// TIA Portal project "Separating_Station" (V15.1)

(* hardware
DEVICE "S7-1200 station_1"  S7-1200 Station
   slot 0: "Rack_0"  S7-1200 Rack  Rack  V1.0
   slot 1: "PLC_1"  CPU 1212C AC/DC/Rly  6ES7 212-1BE40-0XB0  V4.3
*)

// ===== PLC "PLC_1"  CPU 1212C AC/DC/Rly =====

VAR_GLOBAL   // PLC tag table "Default tag table"
   "System_Byte" AT %MB1 : Byte;
   "FirstScan" AT %M1.0 : Bool;
   "DiagStatusUpdate" AT %M1.1 : Bool;
   "AlwaysTRUE" AT %M1.2 : Bool;
   "AlwaysFALSE" AT %M1.3 : Bool;
   "Clock_Byte" AT %MB0 : Byte;
   "Clock_10Hz" AT %M0.0 : Bool;
   "Clock_5Hz" AT %M0.1 : Bool;
   "Clock_2.5Hz" AT %M0.2 : Bool;
   "Clock_2Hz" AT %M0.3 : Bool;
   "Clock_1.25Hz" AT %M0.4 : Bool;
   "Clock_1Hz" AT %M0.5 : Bool;
   "Clock_0.625Hz" AT %M0.6 : Bool;
   "Clock_0.5Hz" AT %M0.7 : Bool;
   "Start" AT %I21.0 : Bool;
   "Stop" AT %I21.1 : Bool;
   "Entry_Conveyor_1" AT %Q20.0 : Bool;
   "SQ_Pusher_1_Front" AT %I20.2 : Bool;
   "SQ_Pusher_1_Back" AT %I20.3 : Bool;
   "Vision_Sensor_1" AT %IW100 : Int;
   "Vision_Sensor_2" AT %IW102 : Int;
   "Entry_Conveyor_2" AT %Q20.1 : Bool;
   "SQ_Pusher_2_Back" AT %I20.6 : Bool;
   "SQ_1" AT %I20.0 : Bool;
   "SQ_2" AT %I20.1 : Bool;
   "Conveyor_1" AT %Q20.2 : Bool;
   "Conveyor_2" AT %Q20.3 : Bool;
   "At_Pusher_1_Exit" AT %I20.4 : Bool;
   "At_Pusher_2_Exit" AT %I20.7 : Bool;
   "Pusher_1" AT %Q20.4 : Bool;
   "Pusher_2" AT %Q20.5 : Bool;
   "SQ_Pusher_2_Front" AT %I20.5 : Bool;
   "Tag_2" AT %I21.2 : Bool;
END_VAR

DATA_BLOCK "Ist_Separating_Station"   // DB1
{ S7_Optimized_Access := 'TRUE' }
AUTHOR : Rackso
VERSION : 0.1
// stored: InstanceOfName Separating_Station
"Separating_Station"
BEGIN
END_DATA_BLOCK

DATA_BLOCK "Edge"   // DB3
{ S7_Optimized_Access := 'TRUE' }
AUTHOR : Rackso
VERSION : 0.1
   VAR
      Negative_Edge : Array[0..15] of Bool;
      Positve_Edge : Array[0..15] of Bool;
   END_VAR
BEGIN
END_DATA_BLOCK

FUNCTION_BLOCK "Separating_Station"   // FB2, LAD
{ S7_Optimized_Access := 'TRUE' }
AUTHOR : Rackso
VERSION : 0.1
   VAR_INPUT
      Sensor_1 : Bool;   // At "Entry conveyor_1" exit
      Sensor_2 : Bool;   // At "Entry conveyor_2" exit
      Pusher_1_front : Bool;   // Extended pusher_1
      Pusher_1_back : Bool;   // Retracted pusher_1
      At_pusher_1_exit : Bool;   // Counter_1
      Pusher_2_front : Bool;   // Extended pusher_2
      Pusher_2_back : Bool;   // Retracted pusher_2
      At_pusher_2_exit : Bool;   // Counter_2
      Start : Bool;
      Stop : Bool;
      FactoryIO_Running : Bool;
      EM_Stop : Bool;
      PEW_Vision_sensor_1 : Int;   // Recognizes raw material "colors" 1=blue, 4=green
      PEW_Vision_sensor_2 : Int;   // Recognizes raw material "colors" 1=blue, 4=green
   END_VAR
   VAR_OUTPUT
      Entry_conveyor_1 : Bool;
      Entry_conveyor_2 : Bool;
      Conveyor_1 : Bool;
      Conveyor_2 : Bool;
      Pusher_1 : Bool;
      Pusher_2 : Bool;
      Emiter_1 : Bool;
      Emiter_2 : Bool;
      Start_light : Bool;
      Stop_light : Bool;
      Reset_light : Bool;
      Counter_1 : Bool;
      Counter_2 : Bool;
   END_VAR
   VAR
      Run_Process : Bool;
      X_Sensor_1 : Bool;
      X_Sensor_2 : Bool;
      Event_1 : Bool;
      X_At_Pusher_1_Exit : Bool;
      Aux_1 : Bool;
      Aux_2 : Bool;
      Event_2 : Bool;
      Event_3 : Bool;
      Event_4 : Bool;
      X_Pusher_1_Back : Bool;
      X_Pusher_2_Back : Bool;
      Event_5 : Bool;
      Event_6 : Bool;
      Event_7 : Bool;
      X_At_Pusher_2_Exit : Bool;
      Aux_Retract_1 : Bool;
      Y1 : Bool;
      Y2 : Bool;
      Aux_Retract_2 : Bool;
      Y3 : Bool;
      Aux_Retract_3 : Bool;
      Aux_1_Conveyor : Bool;
      EN_1_Conveyor_1 : Bool;
      CZ1 : Bool;
      EN_1_Conveyor_2 : Bool;
      Aux_2_Conveyor : Bool;
      EN_2_Conveyor_1 : Bool;
      CZ2 : Bool;
      EN_2_Conveyor_2 : Bool;
      Aux_3_Conveyor : Bool;
      CZ3 : Bool;
      EN_3_Conveyor_1 : Bool;
      EN_3_Conveyor_2 : Bool;
      CZ4 : Bool;
      EN_4_Conveyor_1 : Bool;
      EN_4_Conveyor_2 : Bool;
      Event_8 : Bool;
      Aux_Pusher_1 : Bool;
      Aux_Pusher_2 : Bool;
   END_VAR
   VAR_TEMP   // added for the SCL form of the ladder/FBD networks
      _w1 : Bool;
      _w2 : Bool;
      _w3 : Bool;
      _w4 : Bool;
      _w5 : Bool;
      _w6 : Bool;
      _w7 : Bool;
      _w8 : Bool;
      _w9 : Bool;
      _w10 : Bool;
      _w11 : Bool;
      _w12 : Bool;
      _w13 : Bool;
   END_VAR
BEGIN

REGION Network 1: Start Process
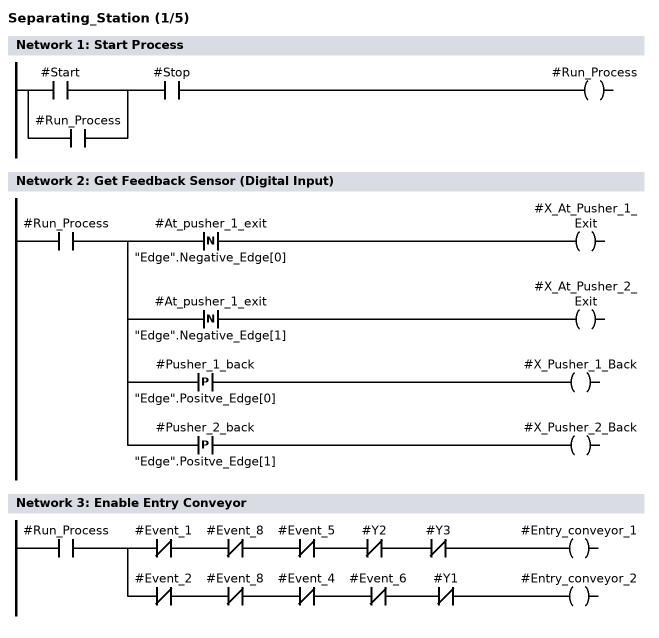
   RUNG wire#powerrail
      Contact( #Start )
      wire#w1
      Contact( #Stop )
      Coil( #Run_Process )
   END_RUNG
   RUNG wire#powerrail
      Contact( #Run_Process )
   END_RUNG wire#w1
   // the same network as SCL:
   #Run_Process := (#Start OR #Run_Process) AND #Stop;
END_REGION

REGION Network 2: Get Feedback Sensor (Digital Input)
   RUNG wire#powerrail
      Contact( #Run_Process )
      wire#w1
      N_Contact(operand := #At_pusher_1_exit, bit := "Edge".Negative_Edge[0])
      Coil( #X_At_Pusher_1_Exit )
   END_RUNG
   RUNG wire#w1
      N_Contact(operand := #At_pusher_1_exit, bit := "Edge".Negative_Edge[1])
      Coil( #X_At_Pusher_2_Exit )
   END_RUNG
   RUNG wire#w1
      P_Contact(operand := #Pusher_1_back, bit := "Edge".Positve_Edge[0])
      Coil( #X_Pusher_1_Back )
   END_RUNG
   RUNG wire#w1
      P_Contact(operand := #Pusher_2_back, bit := "Edge".Positve_Edge[1])
      Coil( #X_Pusher_2_Back )
   END_RUNG
   // the same network as SCL:
   #_w1 := #Run_Process AND NOT #At_pusher_1_exit AND "Edge".Negative_Edge[0];   // falling edge of #At_pusher_1_exit
   "Edge".Negative_Edge[0] := #At_pusher_1_exit;
   #X_At_Pusher_1_Exit := #_w1;
   #_w2 := #Run_Process AND NOT #At_pusher_1_exit AND "Edge".Negative_Edge[1];   // falling edge of #At_pusher_1_exit
   "Edge".Negative_Edge[1] := #At_pusher_1_exit;
   #X_At_Pusher_2_Exit := #_w2;
   #_w3 := #Run_Process AND #Pusher_1_back AND NOT "Edge".Positve_Edge[0];   // rising edge of #Pusher_1_back
   "Edge".Positve_Edge[0] := #Pusher_1_back;
   #X_Pusher_1_Back := #_w3;
   #_w4 := #Run_Process AND #Pusher_2_back AND NOT "Edge".Positve_Edge[1];   // rising edge of #Pusher_2_back
   "Edge".Positve_Edge[1] := #Pusher_2_back;
   #X_Pusher_2_Back := #_w4;
END_REGION

REGION Network 3: Enable Entry Conveyor
   RUNG wire#powerrail
      Contact( #Run_Process )
      wire#w1
      I_Contact( #Event_1 )
      I_Contact( #Event_8 )
      I_Contact( #Event_5 )
      I_Contact( #Y2 )
      I_Contact( #Y3 )
      Coil( #Entry_conveyor_1 )
   END_RUNG
   RUNG wire#w1
      I_Contact( #Event_2 )
      I_Contact( #Event_8 )
      I_Contact( #Event_4 )
      I_Contact( #Event_6 )
      I_Contact( #Y1 )
      Coil( #Entry_conveyor_2 )
   END_RUNG
   // the same network as SCL:
   #Entry_conveyor_1 := #Run_Process AND NOT #Event_1 AND NOT #Event_8 AND NOT #Event_5 AND NOT #Y2 AND NOT #Y3;
   #Entry_conveyor_2 := #Run_Process AND NOT #Event_2 AND NOT #Event_8 AND NOT #Event_4 AND NOT #Event_6 AND NOT #Y1;
END_REGION

REGION Network 4: Get Feedback Sensor Analog Input)
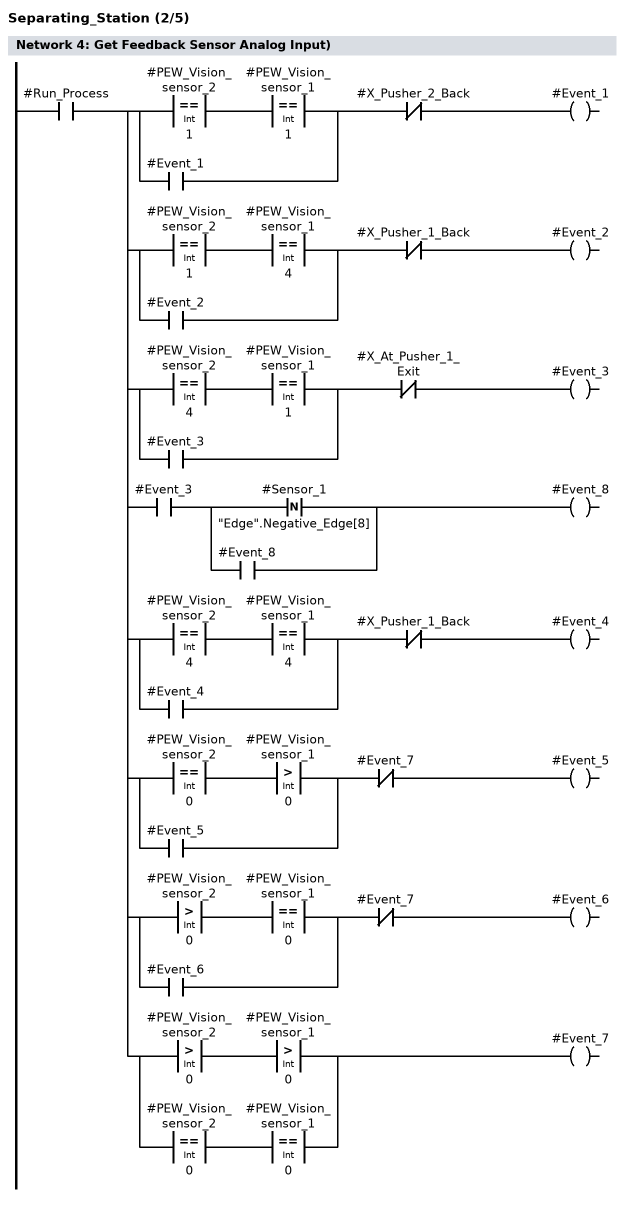
   RUNG wire#powerrail
      Contact( #Run_Process )
      wire#w1
      { S7_Templates := "SrcType := Int" } EQ_Contact(in1 := #PEW_Vision_sensor_2, in2 := 1)
      { S7_Templates := "SrcType := Int" } EQ_Contact(in1 := #PEW_Vision_sensor_1, in2 := 1)
      wire#w2
      I_Contact( #X_Pusher_2_Back )
      Coil( #Event_1 )
   END_RUNG
   RUNG wire#w1
      Contact( #Event_1 )
   END_RUNG wire#w2
   RUNG wire#w1
      { S7_Templates := "SrcType := Int" } EQ_Contact(in1 := #PEW_Vision_sensor_2, in2 := 1)
      { S7_Templates := "SrcType := Int" } EQ_Contact(in1 := #PEW_Vision_sensor_1, in2 := 4)
      wire#w3
      I_Contact( #X_Pusher_1_Back )
      Coil( #Event_2 )
   END_RUNG
   RUNG wire#w1
      Contact( #Event_2 )
   END_RUNG wire#w3
   RUNG wire#w1
      { S7_Templates := "SrcType := Int" } EQ_Contact(in1 := #PEW_Vision_sensor_2, in2 := 4)
      { S7_Templates := "SrcType := Int" } EQ_Contact(in1 := #PEW_Vision_sensor_1, in2 := 1)
      wire#w4
      I_Contact( #X_At_Pusher_1_Exit )
      Coil( #Event_3 )
   END_RUNG
   RUNG wire#w1
      Contact( #Event_3 )
   END_RUNG wire#w4
   RUNG wire#w1
      Contact( #Event_3 )
      wire#w5
      N_Contact(operand := #Sensor_1, bit := "Edge".Negative_Edge[8])
      wire#w6
      Coil( #Event_8 )
   END_RUNG
   RUNG wire#w5
      Contact( #Event_8 )
   END_RUNG wire#w6
   RUNG wire#w1
      { S7_Templates := "SrcType := Int" } EQ_Contact(in1 := #PEW_Vision_sensor_2, in2 := 4)
      { S7_Templates := "SrcType := Int" } EQ_Contact(in1 := #PEW_Vision_sensor_1, in2 := 4)
      wire#w7
      I_Contact( #X_Pusher_1_Back )
      Coil( #Event_4 )
   END_RUNG
   RUNG wire#w1
      Contact( #Event_4 )
   END_RUNG wire#w7
   RUNG wire#w1
      { S7_Templates := "SrcType := Int" } EQ_Contact(in1 := #PEW_Vision_sensor_2, in2 := 0)
      { S7_Templates := "SrcType := Int" } GT_Contact(in1 := #PEW_Vision_sensor_1, in2 := 0)
      wire#w8
      I_Contact( #Event_7 )
      Coil( #Event_5 )
   END_RUNG
   RUNG wire#w1
      Contact( #Event_5 )
   END_RUNG wire#w8
   RUNG wire#w1
      { S7_Templates := "SrcType := Int" } GT_Contact(in1 := #PEW_Vision_sensor_2, in2 := 0)
      { S7_Templates := "SrcType := Int" } EQ_Contact(in1 := #PEW_Vision_sensor_1, in2 := 0)
      wire#w9
      I_Contact( #Event_7 )
      Coil( #Event_6 )
   END_RUNG
   RUNG wire#w1
      Contact( #Event_6 )
   END_RUNG wire#w9
   RUNG wire#w1
      { S7_Templates := "SrcType := Int" } GT_Contact(in1 := #PEW_Vision_sensor_2, in2 := 0)
      { S7_Templates := "SrcType := Int" } GT_Contact(in1 := #PEW_Vision_sensor_1, in2 := 0)
      wire#w10
      Coil( #Event_7 )
   END_RUNG
   RUNG wire#w1
      { S7_Templates := "SrcType := Int" } EQ_Contact(in1 := #PEW_Vision_sensor_2, in2 := 0)
      { S7_Templates := "SrcType := Int" } EQ_Contact(in1 := #PEW_Vision_sensor_1, in2 := 0)
   END_RUNG wire#w10
   // the same network as SCL:
   #Event_1 := #Run_Process AND (((#PEW_Vision_sensor_2 = 1) AND (#PEW_Vision_sensor_1 = 1)) OR #Event_1) AND NOT #X_Pusher_2_Back;
   #Event_2 := #Run_Process AND (((#PEW_Vision_sensor_2 = 1) AND (#PEW_Vision_sensor_1 = 4)) OR #Event_2) AND NOT #X_Pusher_1_Back;
   #Event_3 := #Run_Process AND (((#PEW_Vision_sensor_2 = 4) AND (#PEW_Vision_sensor_1 = 1)) OR #Event_3) AND NOT #X_At_Pusher_1_Exit;
   #_w1 := #Run_Process AND #Event_3 AND NOT #Sensor_1 AND "Edge".Negative_Edge[8];   // falling edge of #Sensor_1
   "Edge".Negative_Edge[8] := #Sensor_1;
   #Event_8 := #_w1 OR (#Run_Process AND #Event_3 AND #Event_8);
   #Event_4 := #Run_Process AND (((#PEW_Vision_sensor_2 = 4) AND (#PEW_Vision_sensor_1 = 4)) OR #Event_4) AND NOT #X_Pusher_1_Back;
   #Event_5 := #Run_Process AND (((#PEW_Vision_sensor_2 = 0) AND (#PEW_Vision_sensor_1 > 0)) OR #Event_5) AND NOT #Event_7;
   #Event_6 := #Run_Process AND (((#PEW_Vision_sensor_2 > 0) AND (#PEW_Vision_sensor_1 = 0)) OR #Event_6) AND NOT #Event_7;
   #Event_7 := #Run_Process AND (((#PEW_Vision_sensor_2 > 0) AND (#PEW_Vision_sensor_1 > 0)) OR ((#PEW_Vision_sensor_2 = 0) AND (#PEW_Vision_sensor_1 = 0)));
END_REGION

REGION Network 5: Aux Enable Pusher
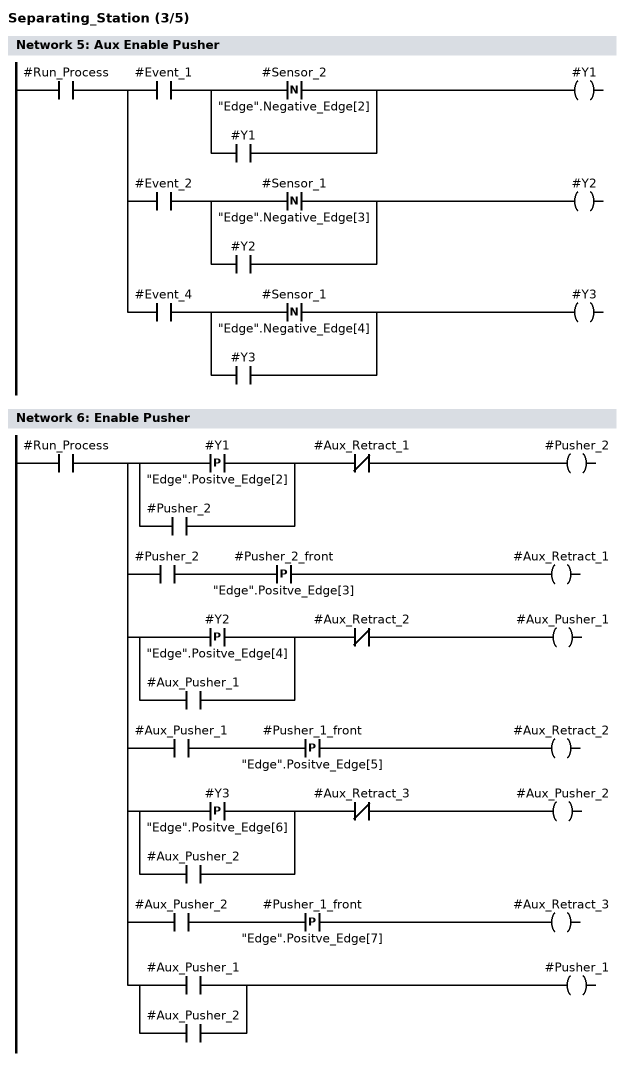
   RUNG wire#powerrail
      Contact( #Run_Process )
      wire#w1
      Contact( #Event_1 )
      wire#w2
      N_Contact(operand := #Sensor_2, bit := "Edge".Negative_Edge[2])
      wire#w3
      Coil( #Y1 )
   END_RUNG
   RUNG wire#w2
      Contact( #Y1 )
   END_RUNG wire#w3
   RUNG wire#w1
      Contact( #Event_2 )
      wire#w4
      N_Contact(operand := #Sensor_1, bit := "Edge".Negative_Edge[3])
      wire#w5
      Coil( #Y2 )
   END_RUNG
   RUNG wire#w4
      Contact( #Y2 )
   END_RUNG wire#w5
   RUNG wire#w1
      Contact( #Event_4 )
      wire#w6
      N_Contact(operand := #Sensor_1, bit := "Edge".Negative_Edge[4])
      wire#w7
      Coil( #Y3 )
   END_RUNG
   RUNG wire#w6
      Contact( #Y3 )
   END_RUNG wire#w7
   // the same network as SCL:
   #_w1 := #Run_Process AND #Event_1 AND NOT #Sensor_2 AND "Edge".Negative_Edge[2];   // falling edge of #Sensor_2
   "Edge".Negative_Edge[2] := #Sensor_2;
   #Y1 := #_w1 OR (#Run_Process AND #Event_1 AND #Y1);
   #_w2 := #Run_Process AND #Event_2 AND NOT #Sensor_1 AND "Edge".Negative_Edge[3];   // falling edge of #Sensor_1
   "Edge".Negative_Edge[3] := #Sensor_1;
   #Y2 := #_w2 OR (#Run_Process AND #Event_2 AND #Y2);
   #_w3 := #Run_Process AND #Event_4 AND NOT #Sensor_1 AND "Edge".Negative_Edge[4];   // falling edge of #Sensor_1
   "Edge".Negative_Edge[4] := #Sensor_1;
   #Y3 := #_w3 OR (#Run_Process AND #Event_4 AND #Y3);
END_REGION

REGION Network 6: Enable Pusher
   RUNG wire#powerrail
      Contact( #Run_Process )
      wire#w1
      P_Contact(operand := #Y1, bit := "Edge".Positve_Edge[2])
      wire#w2
      I_Contact( #Aux_Retract_1 )
      Coil( #Pusher_2 )
   END_RUNG
   RUNG wire#w1
      Contact( #Pusher_2 )
   END_RUNG wire#w2
   RUNG wire#w1
      Contact( #Pusher_2 )
      P_Contact(operand := #Pusher_2_front, bit := "Edge".Positve_Edge[3])
      Coil( #Aux_Retract_1 )
   END_RUNG
   RUNG wire#w1
      P_Contact(operand := #Y2, bit := "Edge".Positve_Edge[4])
      wire#w3
      I_Contact( #Aux_Retract_2 )
      Coil( #Aux_Pusher_1 )
   END_RUNG
   RUNG wire#w1
      Contact( #Aux_Pusher_1 )
   END_RUNG wire#w3
   RUNG wire#w1
      Contact( #Aux_Pusher_1 )
      P_Contact(operand := #Pusher_1_front, bit := "Edge".Positve_Edge[5])
      Coil( #Aux_Retract_2 )
   END_RUNG
   RUNG wire#w1
      P_Contact(operand := #Y3, bit := "Edge".Positve_Edge[6])
      wire#w4
      I_Contact( #Aux_Retract_3 )
      Coil( #Aux_Pusher_2 )
   END_RUNG
   RUNG wire#w1
      Contact( #Aux_Pusher_2 )
   END_RUNG wire#w4
   RUNG wire#w1
      Contact( #Aux_Pusher_2 )
      P_Contact(operand := #Pusher_1_front, bit := "Edge".Positve_Edge[7])
      Coil( #Aux_Retract_3 )
   END_RUNG
   RUNG wire#w1
      Contact( #Aux_Pusher_1 )
      wire#w5
      Coil( #Pusher_1 )
   END_RUNG
   RUNG wire#w1
      Contact( #Aux_Pusher_2 )
   END_RUNG wire#w5
   // the same network as SCL:
   #_w1 := #Run_Process AND #Y1 AND NOT "Edge".Positve_Edge[2];   // rising edge of #Y1
   "Edge".Positve_Edge[2] := #Y1;
   #Pusher_2 := (#_w1 OR (#Run_Process AND #Pusher_2)) AND NOT #Aux_Retract_1;
   #_w2 := #Run_Process AND #Pusher_2 AND #Pusher_2_front AND NOT "Edge".Positve_Edge[3];   // rising edge of #Pusher_2_front
   "Edge".Positve_Edge[3] := #Pusher_2_front;
   #Aux_Retract_1 := #_w2;
   #_w3 := #Run_Process AND #Y2 AND NOT "Edge".Positve_Edge[4];   // rising edge of #Y2
   "Edge".Positve_Edge[4] := #Y2;
   #Aux_Pusher_1 := (#_w3 OR (#Run_Process AND #Aux_Pusher_1)) AND NOT #Aux_Retract_2;
   #_w4 := #Run_Process AND #Aux_Pusher_1 AND #Pusher_1_front AND NOT "Edge".Positve_Edge[5];   // rising edge of #Pusher_1_front
   "Edge".Positve_Edge[5] := #Pusher_1_front;
   #Aux_Retract_2 := #_w4;
   #_w5 := #Run_Process AND #Y3 AND NOT "Edge".Positve_Edge[6];   // rising edge of #Y3
   "Edge".Positve_Edge[6] := #Y3;
   #Aux_Pusher_2 := (#_w5 OR (#Run_Process AND #Aux_Pusher_2)) AND NOT #Aux_Retract_3;
   #_w6 := #Run_Process AND #Aux_Pusher_2 AND #Pusher_1_front AND NOT "Edge".Positve_Edge[7];   // rising edge of #Pusher_1_front
   "Edge".Positve_Edge[7] := #Pusher_1_front;
   #Aux_Retract_3 := #_w6;
   #Pusher_1 := #Run_Process AND (#Aux_Pusher_1 OR #Aux_Pusher_2);
END_REGION

REGION Network 7: Aux Enbale Conveyor
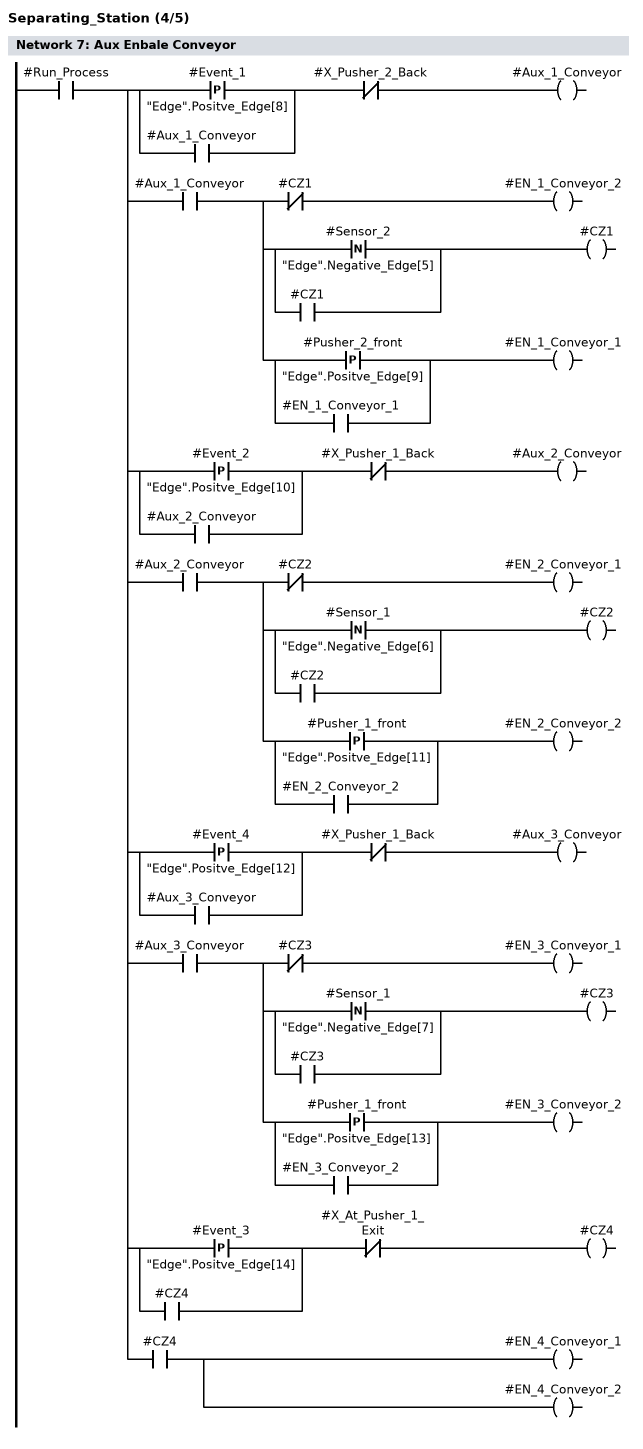
   RUNG wire#powerrail
      Contact( #Run_Process )
      wire#w1
      P_Contact(operand := #Event_1, bit := "Edge".Positve_Edge[8])
      wire#w2
      I_Contact( #X_Pusher_2_Back )
      Coil( #Aux_1_Conveyor )
   END_RUNG
   RUNG wire#w1
      Contact( #Aux_1_Conveyor )
   END_RUNG wire#w2
   RUNG wire#w1
      Contact( #Aux_1_Conveyor )
      wire#w3
      I_Contact( #CZ1 )
      Coil( #EN_1_Conveyor_2 )
   END_RUNG
   RUNG wire#w3
      N_Contact(operand := #Sensor_2, bit := "Edge".Negative_Edge[5])
      wire#w4
      Coil( #CZ1 )
   END_RUNG
   RUNG wire#w3
      Contact( #CZ1 )
   END_RUNG wire#w4
   RUNG wire#w3
      P_Contact(operand := #Pusher_2_front, bit := "Edge".Positve_Edge[9])
      wire#w5
      Coil( #EN_1_Conveyor_1 )
   END_RUNG
   RUNG wire#w3
      Contact( #EN_1_Conveyor_1 )
   END_RUNG wire#w5
   RUNG wire#w1
      P_Contact(operand := #Event_2, bit := "Edge".Positve_Edge[10])
      wire#w6
      I_Contact( #X_Pusher_1_Back )
      Coil( #Aux_2_Conveyor )
   END_RUNG
   RUNG wire#w1
      Contact( #Aux_2_Conveyor )
   END_RUNG wire#w6
   RUNG wire#w1
      Contact( #Aux_2_Conveyor )
      wire#w7
      I_Contact( #CZ2 )
      Coil( #EN_2_Conveyor_1 )
   END_RUNG
   RUNG wire#w7
      N_Contact(operand := #Sensor_1, bit := "Edge".Negative_Edge[6])
      wire#w8
      Coil( #CZ2 )
   END_RUNG
   RUNG wire#w7
      Contact( #CZ2 )
   END_RUNG wire#w8
   RUNG wire#w7
      P_Contact(operand := #Pusher_1_front, bit := "Edge".Positve_Edge[11])
      wire#w9
      Coil( #EN_2_Conveyor_2 )
   END_RUNG
   RUNG wire#w7
      Contact( #EN_2_Conveyor_2 )
   END_RUNG wire#w9
   RUNG wire#w1
      P_Contact(operand := #Event_4, bit := "Edge".Positve_Edge[12])
      wire#w10
      I_Contact( #X_Pusher_1_Back )
      Coil( #Aux_3_Conveyor )
   END_RUNG
   RUNG wire#w1
      Contact( #Aux_3_Conveyor )
   END_RUNG wire#w10
   RUNG wire#w1
      Contact( #Aux_3_Conveyor )
      wire#w11
      I_Contact( #CZ3 )
      Coil( #EN_3_Conveyor_1 )
   END_RUNG
   RUNG wire#w11
      N_Contact(operand := #Sensor_1, bit := "Edge".Negative_Edge[7])
      wire#w12
      Coil( #CZ3 )
   END_RUNG
   RUNG wire#w11
      Contact( #CZ3 )
   END_RUNG wire#w12
   RUNG wire#w11
      P_Contact(operand := #Pusher_1_front, bit := "Edge".Positve_Edge[13])
      wire#w13
      Coil( #EN_3_Conveyor_2 )
   END_RUNG
   RUNG wire#w11
      Contact( #EN_3_Conveyor_2 )
   END_RUNG wire#w13
   RUNG wire#w1
      P_Contact(operand := #Event_3, bit := "Edge".Positve_Edge[14])
      wire#w14
      I_Contact( #X_At_Pusher_1_Exit )
      Coil( #CZ4 )
   END_RUNG
   RUNG wire#w1
      Contact( #CZ4 )
   END_RUNG wire#w14
   RUNG wire#w1
      Contact( #CZ4 )
      wire#w15
      Coil( #EN_4_Conveyor_1 )
   END_RUNG
   RUNG wire#w15
      Coil( #EN_4_Conveyor_2 )
   END_RUNG
   // the same network as SCL:
   #_w1 := #Run_Process AND #Event_1 AND NOT "Edge".Positve_Edge[8];   // rising edge of #Event_1
   "Edge".Positve_Edge[8] := #Event_1;
   #Aux_1_Conveyor := (#_w1 OR (#Run_Process AND #Aux_1_Conveyor)) AND NOT #X_Pusher_2_Back;
   #_w2 := #Run_Process AND #Aux_1_Conveyor;
   #EN_1_Conveyor_2 := #_w2 AND NOT #CZ1;
   #_w3 := #_w2 AND NOT #Sensor_2 AND "Edge".Negative_Edge[5];   // falling edge of #Sensor_2
   "Edge".Negative_Edge[5] := #Sensor_2;
   #CZ1 := #_w3 OR (#_w2 AND #CZ1);
   #_w4 := #_w2 AND #Pusher_2_front AND NOT "Edge".Positve_Edge[9];   // rising edge of #Pusher_2_front
   "Edge".Positve_Edge[9] := #Pusher_2_front;
   #EN_1_Conveyor_1 := #_w4 OR (#_w2 AND #EN_1_Conveyor_1);
   #_w5 := #Run_Process AND #Event_2 AND NOT "Edge".Positve_Edge[10];   // rising edge of #Event_2
   "Edge".Positve_Edge[10] := #Event_2;
   #Aux_2_Conveyor := (#_w5 OR (#Run_Process AND #Aux_2_Conveyor)) AND NOT #X_Pusher_1_Back;
   #_w6 := #Run_Process AND #Aux_2_Conveyor;
   #EN_2_Conveyor_1 := #_w6 AND NOT #CZ2;
   #_w7 := #_w6 AND NOT #Sensor_1 AND "Edge".Negative_Edge[6];   // falling edge of #Sensor_1
   "Edge".Negative_Edge[6] := #Sensor_1;
   #CZ2 := #_w7 OR (#_w6 AND #CZ2);
   #_w8 := #_w6 AND #Pusher_1_front AND NOT "Edge".Positve_Edge[11];   // rising edge of #Pusher_1_front
   "Edge".Positve_Edge[11] := #Pusher_1_front;
   #EN_2_Conveyor_2 := #_w8 OR (#_w6 AND #EN_2_Conveyor_2);
   #_w9 := #Run_Process AND #Event_4 AND NOT "Edge".Positve_Edge[12];   // rising edge of #Event_4
   "Edge".Positve_Edge[12] := #Event_4;
   #Aux_3_Conveyor := (#_w9 OR (#Run_Process AND #Aux_3_Conveyor)) AND NOT #X_Pusher_1_Back;
   #_w10 := #Run_Process AND #Aux_3_Conveyor;
   #EN_3_Conveyor_1 := #_w10 AND NOT #CZ3;
   #_w11 := #_w10 AND NOT #Sensor_1 AND "Edge".Negative_Edge[7];   // falling edge of #Sensor_1
   "Edge".Negative_Edge[7] := #Sensor_1;
   #CZ3 := #_w11 OR (#_w10 AND #CZ3);
   #_w12 := #_w10 AND #Pusher_1_front AND NOT "Edge".Positve_Edge[13];   // rising edge of #Pusher_1_front
   "Edge".Positve_Edge[13] := #Pusher_1_front;
   #EN_3_Conveyor_2 := #_w12 OR (#_w10 AND #EN_3_Conveyor_2);
   #_w13 := #Run_Process AND #Event_3 AND NOT "Edge".Positve_Edge[14];   // rising edge of #Event_3
   "Edge".Positve_Edge[14] := #Event_3;
   #CZ4 := (#_w13 OR (#Run_Process AND #CZ4)) AND NOT #X_At_Pusher_1_Exit;
   #EN_4_Conveyor_1 := #Run_Process AND #CZ4;
   #EN_4_Conveyor_2 := #EN_4_Conveyor_1;
END_REGION

REGION Network 8: Enable Conveyor
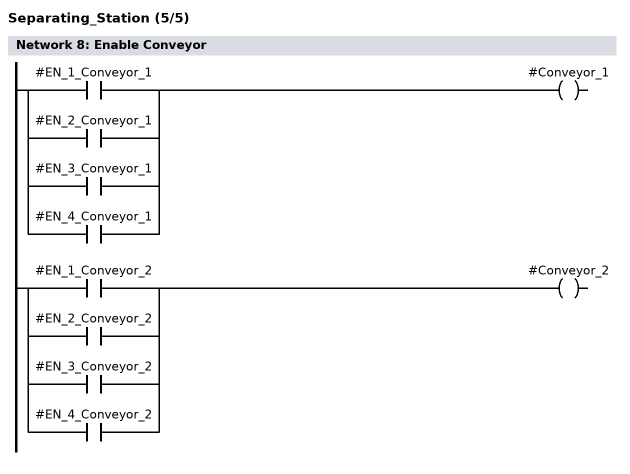
   RUNG wire#powerrail
      Contact( #EN_1_Conveyor_1 )
      wire#w1
      Coil( #Conveyor_1 )
   END_RUNG
   RUNG wire#powerrail
      Contact( #EN_2_Conveyor_1 )
   END_RUNG wire#w1
   RUNG wire#powerrail
      Contact( #EN_3_Conveyor_1 )
   END_RUNG wire#w1
   RUNG wire#powerrail
      Contact( #EN_4_Conveyor_1 )
   END_RUNG wire#w1
   RUNG wire#powerrail
      Contact( #EN_1_Conveyor_2 )
      wire#w2
      Coil( #Conveyor_2 )
   END_RUNG
   RUNG wire#powerrail
      Contact( #EN_2_Conveyor_2 )
   END_RUNG wire#w2
   RUNG wire#powerrail
      Contact( #EN_3_Conveyor_2 )
   END_RUNG wire#w2
   RUNG wire#powerrail
      Contact( #EN_4_Conveyor_2 )
   END_RUNG wire#w2
   // the same network as SCL:
   #Conveyor_1 := #EN_1_Conveyor_1 OR #EN_2_Conveyor_1 OR #EN_3_Conveyor_1 OR #EN_4_Conveyor_1;
   #Conveyor_2 := #EN_1_Conveyor_2 OR #EN_2_Conveyor_2 OR #EN_3_Conveyor_2 OR #EN_4_Conveyor_2;
END_REGION
END_FUNCTION_BLOCK

ORGANIZATION_BLOCK "Main"   // OB1, LAD, ProgramCycle
TITLE = "Main Program Sweep (Cycle)"
{ S7_Optimized_Access := 'TRUE' }
VERSION : 0.1
   VAR_INPUT
      Initial_Call : Bool;   // Initial call of this OB
      Remanence : Bool;   // =True, if remanent data are available
   END_VAR
BEGIN

REGION Network 1
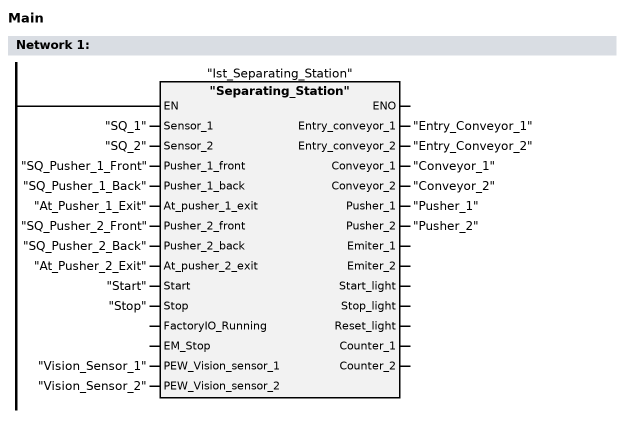
   RUNG wire#powerrail
      "Ist_Separating_Station"(Sensor_1 := "SQ_1", Sensor_2 := "SQ_2", Pusher_1_front := "SQ_Pusher_1_Front", Pusher_1_back := "SQ_Pusher_1_Back", At_pusher_1_exit := "At_Pusher_1_Exit", Pusher_2_front := "SQ_Pusher_2_Front", Pusher_2_back := "SQ_Pusher_2_Back", At_pusher_2_exit := "At_Pusher_2_Exit", Start := "Start", Stop := "Stop", FactoryIO_Running :=, EM_Stop :=, PEW_Vision_sensor_1 := "Vision_Sensor_1", PEW_Vision_sensor_2 := "Vision_Sensor_2", Entry_conveyor_1 => "Entry_Conveyor_1", Entry_conveyor_2 => "Entry_Conveyor_2", Conveyor_1 => "Conveyor_1", Conveyor_2 => "Conveyor_2", Pusher_1 => "Pusher_1", Pusher_2 => "Pusher_2", Emiter_1 =>, Emiter_2 =>, Start_light =>, Stop_light =>, Reset_light =>, Counter_1 =>, Counter_2 =>)
   END_RUNG
   // the same network as SCL:
   "Ist_Separating_Station"(Sensor_1 := "SQ_1",   // "Separating_Station"
                           Sensor_2 := "SQ_2",
                           Pusher_1_front := "SQ_Pusher_1_Front",
                           Pusher_1_back := "SQ_Pusher_1_Back",
                           At_pusher_1_exit := "At_Pusher_1_Exit",
                           Pusher_2_front := "SQ_Pusher_2_Front",
                           Pusher_2_back := "SQ_Pusher_2_Back",
                           At_pusher_2_exit := "At_Pusher_2_Exit",
                           Start := "Start",
                           Stop := "Stop",
                           PEW_Vision_sensor_1 := "Vision_Sensor_1",
                           PEW_Vision_sensor_2 := "Vision_Sensor_2",
                           Entry_conveyor_1 => "Entry_Conveyor_1",
                           Entry_conveyor_2 => "Entry_Conveyor_2",
                           Conveyor_1 => "Conveyor_1",
                           Conveyor_2 => "Conveyor_2",
                           Pusher_1 => "Pusher_1",
                           Pusher_2 => "Pusher_2");
END_REGION
END_ORGANIZATION_BLOCK

// ===== library types =====

// folder: LGF/0 Bit logic operations

FUNCTION_BLOCK "LGF_PulseRelay"   // FB10000, SCL
TITLE = LGF_PulseRelay
{ S7_Optimized_Access := 'TRUE' }
AUTHOR : Siemens_Digital_Industry
FAMILY : LGF
NAME : LGF_PulseRelay
// Pulse relay, Surge relay, Toggle-Flip-Flop, Frequency divider
// Reset is leading / prior to Set or trigger
   VAR_INPUT
      trigger : Bool;   // trigger to toggle output signal, rising edge / trigger signal, rising edge
      set : Bool;   // set output signal. rising edge / set signal. rising edge
      reset : Bool;   // reset signal, rising edge (prior to set) / reset signal, rising edge
   END_VAR
   VAR_OUTPUT
      out : Bool;   // output signal
   END_VAR
   VAR
      statTriggerOld : Bool := false;   // store old value of trigger input / -
      statSetOld : Bool := false;   // store old value of set input / -
      statResetOld : Bool := false;   // store old value of reset input / -
      statOut : Bool := false;   // internal status store to keep the last value in the block / -
   END_VAR
BEGIN
   REGION BLOCK INFO HEADER
     //===============================================================================
     // SIEMENS AG / (c)Copyright 2019
     //-------------------------------------------------------------------------------
     // Title:            LGF_PulseRelay
     // Comment/Function: Pulse relay, Surge relay, Toggle-Flip-Flop, Frequency divider
     //                   Reset is leading / prior to Set or Trigger
     // Library/Family:   LGF (Library General Functions)
     // Author:           Siemens Digital Industry
     // Tested with:      CPU1212C DC/DC/DC FW:V4.2
     // Engineering:      TIA Portal V15.1
     // Restrictions:     ENO not in use, set to true, no error handling
     // Requirements:     PLC (S7-1200 / S7-1500)
     //-------------------------------------------------------------------------------
     // Change log table:
     // Version  | Date       | Expert in charge       | Changes applied
     // 01.00.00 06.06.2015 Siemens Industry Online Support
     //                     First released version
     // 01.00.01 02.01.2017 Siemens Industry Online Support
     //                     Upgrade: TIA V14 Update 1
     // 01.00.02 02.01.2017 Siemens Industry Online Support
     //                     Comment correction                  
     // 01.00.03 17.08.2018 Siemens Industry Online Support
     //                     Upgrade: TIA V15 Update 2
     // 01.00.04 23.11.2018 Siemens Industry Online Support
     //                     Upgrade: TIA V15.1
     // 01.00.05 24.05.2019 Siemens Industry Presale Support
     //                     Refactoring and performance improvment
     //                     add eno handling
     // 03.00.00 23.04.2020 Siemens Industry Support
     //                     Set version to V3.0.0, harmonize the version of the whole library
     //===============================================================================
   END_REGION

   REGION PROGRAM LOGIC
     REGION toggle output
       // Scan for rising edge "trigger"  - toggle static Output
       IF #trigger AND NOT #statTriggerOld THEN
         // toggle static output memory
         #statOut := NOT #statOut;
       END_IF;
       // store trigger input for edge dedection
       #statTriggerOld := #trigger;
     END_REGION

     REGION set output
       // Scan for rising edge "set" - static Output: set
       IF #set AND NOT #statSetOld THEN
         // set static output memory
         #statOut := TRUE;
       END_IF;
       // store set input for edge dedection
       #statSetOld := #set;
     END_REGION

     REGION reset output    
       // Scan for rising edge "reset" - static Output: reset
       IF #reset AND NOT #statResetOld THEN
         // store trigger input for edge dedection
         #statOut := FALSE;
       END_IF;
       // store reset input for edge dedection
       #statResetOld := #reset;
     END_REGION
   END_REGION

   REGION OUTPUTS
     // write the Output value
     #out := #statOut;
     // no error handling needed
     ENO := TRUE;
   END_REGION
END_FUNCTION_BLOCK

FUNCTION "LGF_BitSet" : DWord   // FC10078, SCL
TITLE = CADD / LGF_BitSet
{ S7_Optimized_Access := 'TRUE' }
AUTHOR : SiemensSIMATICSystemsSupport
FAMILY : LGF
NAME : LGF_BitSet
// this function add two complex numbers
// 
// uses: COMPLEX [UDT2]
// Set bit in elementary datatype - DWord
// can be used for Word and Byte as well, by convert
// the passed paramter and the result using for e.g. Dword_to_Byte
   VAR_INPUT
      value : DWord;   // tag where the bit has to be set
      bitNo : USInt;   // bit number to set in "value" paramter
   END_VAR
   // Ret_Val : tag with set bit
   VAR CONSTANT
      TRUE_BOOL_BIT : DWord := 16#0001;   // Just one bit which is true, to shift in Dword for masking
      MAX_NO_OF_BITS : USInt := 32;   // Maximum bits in a DWord = 32
   END_VAR
BEGIN
   REGION BLOCK INFO HEADER
     //===============================================================================
     // SIEMENS AG / (c)Copyright 2019
     //-------------------------------------------------------------------------------
     // Title:            LGF_BitSet
     // Comment/Function: Set bit in elementary datatype - DWord
     //                   cam be used for Word and Byte as well, by convert
     //                   the passed paramter and the result using for e.g. Dword_to_Byte
     // Library/Family:   LGF (Library General Functions)
     // Author:           Siemens Digital Industry
     // Tested with:      CPU1212C DC/DC/DC FW:V4.2
     // Engineering:      TIA Portal V15.1
     // Restrictions:     ENO not in use, set to true, no error handling
     // Requirements:     PLC (S7-1200 / S7-1500)
     //-------------------------------------------------------------------------------
     // Change log table:
     // Version  | Date       | Expert in charge         | Changes applied
     // 01.00.00 | 06.06.2015 | Siemens Industry Support | first release
     // 03.00.00 | 23.04.2020 | Siemens Industry Support | Set version to V3.0.0
     //                         harmonize the version of the whole library
     //===============================================================================
   END_REGION

   REGION Logic
     // set the bit in tag
     // shift one true bit into given position
     // concatenate value then with OR will result in the previous value and the set bit in position
     #LGF_BitSet := #value OR SHL(IN := #TRUE_BOOL_BIT, N := (#bitNo MOD #MAX_NO_OF_BITS));

     // no error handling needed
     ENO := TRUE;
   END_REGION
END_FUNCTION